// TIA Portal project "2020-10-30_TestMotoreNO_OK" (V16)

(* hardware
DEVICE "S7-1200 station_1"  S7-1200 Station
   slot 0: "Telaio di montaggio_0"  Rack  V1.0
   slot 1: "PLC_1"  CPU 1215C DC/DC/DC  6ES7 215-1AG40-0XB0  V4.2
*)

// ===== PLC "PLC_1"  CPU 1215C DC/DC/DC =====

VAR_GLOBAL   // PLC tag table "Tabella delle variabili standard"
   "finecorsa_NC" AT %I0.0 : Bool;
   "Presenza_tensione_NA" AT %I0.1 : Bool;
   "Ventilatore_motore_NA" AT %I0.3 : Bool;
   "Start_NA" AT %I0.5 : Bool;
   "Stop_NC" AT %I0.6 : Bool;
   "Allarme_NC" AT %I0.2 : Bool;
   "Ripristino_NA" AT %I0.7 : Bool;
   "Sensore termico mot_NA" AT %I0.4 : Bool;
   "Motore" AT %Q0.0 : Bool;
   "Allarme_mem" AT %Q0.1 : Bool;
   "M_IB0_NCNA" AT %MB0 : Byte;
   "Finecorsa" AT %M0.0 : Bool;
   "Presenza tensione" AT %M0.1 : Bool;
   "Ventilatore motore" AT %M0.3 : Bool;
   "Start" AT %M0.5 : Bool;
   "Stop" AT %M0.6 : Bool;
   "Allarme" AT %M0.2 : Bool;
   "Ripristino" AT %M0.7 : Bool;
   "Sempre_vera" AT %M6.0 : Bool;
   "Ingressi" AT %IB0 : Byte;
   "XXX_Start_old" AT %M1.5 : Bool;
   "XXX_Ripristino_old" AT %M1.7 : Bool;
   "Sensore_termico_mot" AT %M0.4 : Bool;
   "Guasto_ventil" AT %Q0.2 : Bool;
   "Allarme_gen" AT %Q0.3 : Bool;
   "Arresto_anomalo" AT %Q0.4 : Bool;
   "XXX2_ripristino_old" AT %M2.7 : Bool;
   "XXX2_start_old" AT %M2.5 : Bool;
END_VAR

VAR_GLOBAL CONSTANT   // PLC tag table "Tabella delle variabili standard"
   "Maschera NCNA" : Byte := 2#01000101;
END_VAR

ORGANIZATION_BLOCK "Main"   // OB1, LAD, ProgramCycle
TITLE = "Main Program Sweep (Cycle)"
{ S7_Optimized_Access := 'TRUE' }
VERSION : 0.1
// Programma c_mot_all_guast_arresto anomalo
// Step:
// a_ gestione start (I0.5 NA) Stop (I0.6 NC) motore (Q0.0) se presenza tensione (I0.1), con ventilatore acceso (I0.3 NA), logica di finecorsa di sicurezza (i0.0, NC) per arresto motore e sensore termico motore non intervenuto (I0.4 NA). Gestione Lampada Allarme (Q0.1) con memorizzazione ripristino e rientro (Allarme I0.2, NC, Ripristino I0.7 NA)
// 
// b_ funzionalità a, più gestione guasto ventilazione motore (Q0.2) se ventilatore acceso (I0.3 NA) e sensore termico motore intervenuto (I0.4 NA) con motore in movimento. 
// 
// c_ aggiunta gestione Allarme_generale (Q0.3), comprensivo di lampada allarme e guasto ventilatore, e aggiunta arresto motore anomalo (Q0.4) che si accende se il motore viene arrestato da situazioni non corrette (intervento finecorsa di sicurezza o allarme o caduta presenza tensione). Il pulsante Start viene utilizzato per resettare l'anomalia che è di sola segnalazione e non necessita di ripristino
// 
// ISTRUZIONI 
// *Si realizzi un programma di controllo per un motore. Il motore è azionato da un pulsante di Start e fermato dal pulsante di Stop.
// 
// Mappare ingressi NA/NC in memoria, in modo da lavorare in logica vera nel programma.
// Il motore parte se ho tensione, premo start e non sono in condizioni anomale per le quali il motore deve stare fermo.
// Il motore deve fermarsi se c'è un allarme o premo stop o finecorsa o se cade la tensione.
// Si consideri il fermo motore anche in caso di guasto ventilatore e e sensore termico
// 
// NOTA: Gestire incastro Pulsanti e motore
// 
// I0.0	Finecorsa_NC
// I0.1	Presenza_Tensione_NA
// I0.2	Allarme_NC	
// I0.3	Ventilatore_Motore_NA
// I0.4	Sensore_Termico_Motore_NA
// I0.5	Start_NA
// I0.6	Stop_NC
// I0.7	Ripristino_NA
// 
// Q0.0	Motore			   Motore avviato
// Q0.1	Lampada_Allarme	   Segnalazione allarme con memorizzazione ripristino e rientro
// Q0.2    Sirena guasto Ventilatore     Se Motore ON e Ventilatore ON e Sensore Termico ON allora Q0.3    Allarme_generale      Si setta in Presenza di Allarmemem o si guasto Ventil e si resetta con Ripristino
// Q0.4    Arresto motore anomalo     Si accende se il motore viene arrestato da situazioni non corrette (intervento finecorsa di sicurezza o allarme o caduta presenza tensione). Il pulsante Start viene utilizzato per resettare l'anomalia che è di sola segnalazione e non necessita di ripristino
   VAR_TEMP   // added for the SCL form of the ladder/FBD networks
      _w1 : Bool;
   END_VAR
BEGIN

REGION Network 1: Bit Sempre_vero
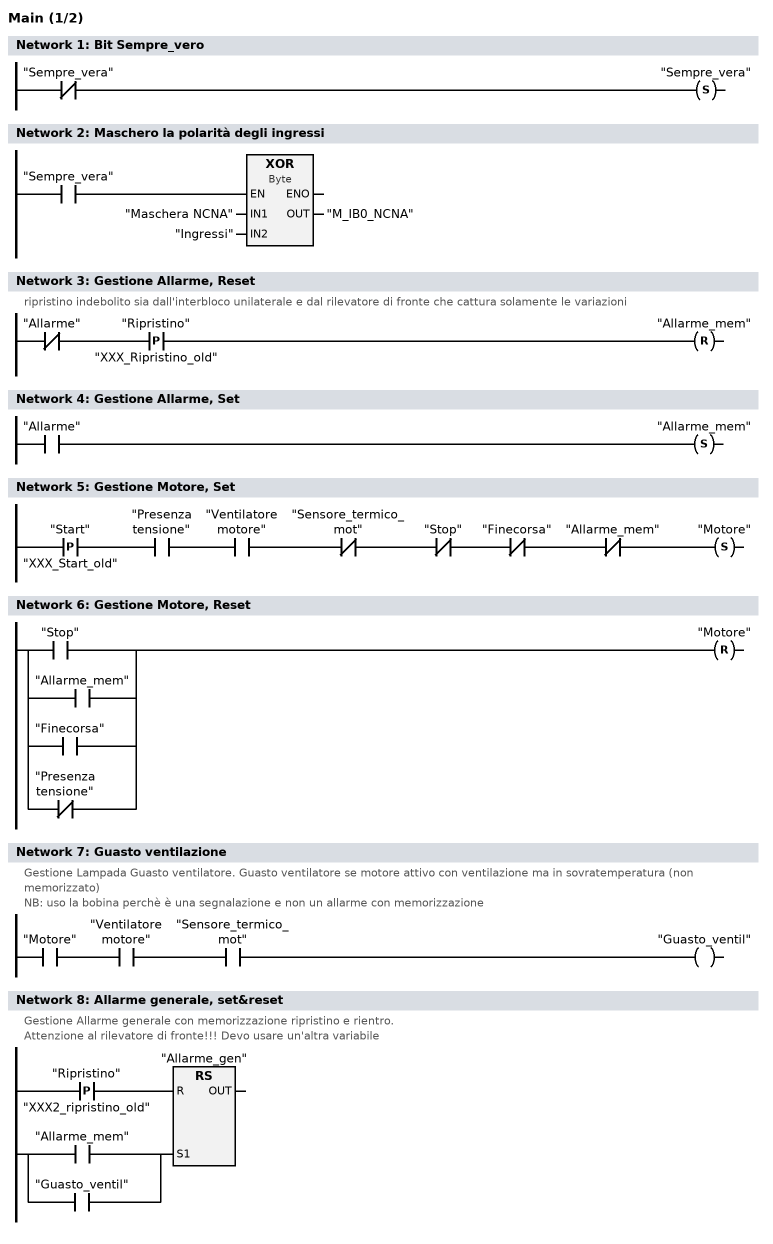
   RUNG wire#powerrail
      I_Contact( "Sempre_vera" )
      S_Coil( "Sempre_vera" )
   END_RUNG
   // the same network as SCL:
   IF NOT "Sempre_vera" THEN "Sempre_vera" := TRUE; END_IF;
END_REGION

REGION Network 2: Maschero la polarità degli ingressi
   IF "Sempre_vera" THEN "M_IB0_NCNA" := "Maschera NCNA" XOR "Ingressi"; END_IF;
END_REGION

REGION Network 3: Gestione Allarme, Reset
   // ripristino indebolito sia dall'interbloco unilaterale e dal rilevatore di fronte che cattura solamente le variazioni
   RUNG wire#powerrail
      I_Contact( "Allarme" )
      P_Contact(operand := "Ripristino", bit := "XXX_Ripristino_old")
      R_Coil( "Allarme_mem" )
   END_RUNG
   // the same network as SCL:
   #_w1 := NOT "Allarme" AND "Ripristino" AND NOT "XXX_Ripristino_old";   // rising edge of "Ripristino"
   "XXX_Ripristino_old" := "Ripristino";
   IF #_w1 THEN "Allarme_mem" := FALSE; END_IF;
END_REGION

REGION Network 4: Gestione Allarme, Set
   RUNG wire#powerrail
      Contact( "Allarme" )
      S_Coil( "Allarme_mem" )
   END_RUNG
   // the same network as SCL:
   IF "Allarme" THEN "Allarme_mem" := TRUE; END_IF;
END_REGION

REGION Network 5: Gestione Motore, Set
   RUNG wire#powerrail
      P_Contact(operand := "Start", bit := "XXX_Start_old")
      Contact( "Presenza tensione" )
      Contact( "Ventilatore motore" )
      I_Contact( "Sensore_termico_mot" )
      I_Contact( "Stop" )
      I_Contact( "Finecorsa" )
      I_Contact( "Allarme_mem" )
      S_Coil( "Motore" )
   END_RUNG
   // the same network as SCL:
   #_w1 := "Start" AND NOT "XXX_Start_old";   // rising edge of "Start"
   "XXX_Start_old" := "Start";
   IF #_w1 AND "Presenza tensione" AND "Ventilatore motore" AND NOT "Sensore_termico_mot" AND NOT "Stop" AND NOT "Finecorsa" AND NOT "Allarme_mem" THEN
       "Motore" := TRUE;
   END_IF;
END_REGION

REGION Network 6: Gestione Motore, Reset
   RUNG wire#powerrail
      Contact( "Stop" )
      wire#w1
      R_Coil( "Motore" )
   END_RUNG
   RUNG wire#powerrail
      Contact( "Allarme_mem" )
   END_RUNG wire#w1
   RUNG wire#powerrail
      Contact( "Finecorsa" )
   END_RUNG wire#w1
   RUNG wire#powerrail
      I_Contact( "Presenza tensione" )
   END_RUNG wire#w1
   // the same network as SCL:
   IF "Stop" OR "Allarme_mem" OR "Finecorsa" OR NOT "Presenza tensione" THEN "Motore" := FALSE; END_IF;
END_REGION

REGION Network 7: Guasto ventilazione
   // Gestione Lampada Guasto ventilatore. Guasto ventilatore se motore attivo con ventilazione ma in sovratemperatura (non memorizzato)
   // NB: uso la bobina perchè è una segnalazione e non un allarme con memorizzazione
   RUNG wire#powerrail
      Contact( "Motore" )
      Contact( "Ventilatore motore" )
      Contact( "Sensore_termico_mot" )
      Coil( "Guasto_ventil" )
   END_RUNG
   // the same network as SCL:
   "Guasto_ventil" := "Motore" AND "Ventilatore motore" AND "Sensore_termico_mot";
END_REGION

REGION Network 8: Allarme generale, set&reset
   // Gestione Allarme generale con memorizzazione ripristino e rientro.
   // Attenzione al rilevatore di fronte!!! Devo usare un'altra variabile
   RUNG wire#powerrail
      P_Contact(operand := "Ripristino", bit := "XXX2_ripristino_old")
      S_RS(operand := "Allarme_gen", s1 := wire#w1)
   END_RUNG
   RUNG wire#powerrail
      Contact( "Allarme_mem" )
   END_RUNG wire#w1
   RUNG wire#powerrail
      Contact( "Guasto_ventil" )
   END_RUNG wire#w1
   // the same network as SCL:
   #_w1 := "Ripristino" AND NOT "XXX2_ripristino_old";   // rising edge of "Ripristino"
   "XXX2_ripristino_old" := "Ripristino";
   IF #_w1 THEN
       "Allarme_gen" := FALSE;   // RS flip-flop
   END_IF;
   IF "Allarme_mem" OR "Guasto_ventil" THEN "Allarme_gen" := TRUE; END_IF;
END_REGION

REGION Network 9: Condizione arresto anomalo, reset
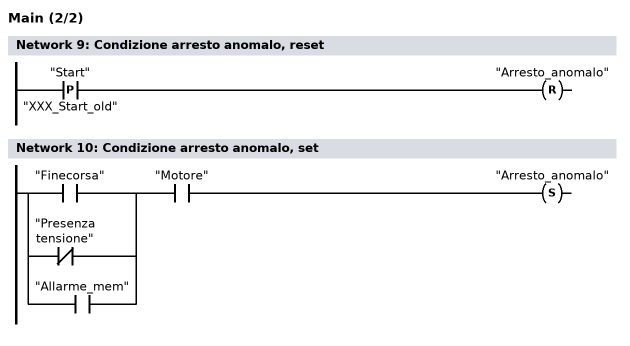
   RUNG wire#powerrail
      P_Contact(operand := "Start", bit := "XXX_Start_old")
      R_Coil( "Arresto_anomalo" )
   END_RUNG
   // the same network as SCL:
   #_w1 := "Start" AND NOT "XXX_Start_old";   // rising edge of "Start"
   "XXX_Start_old" := "Start";
   IF #_w1 THEN "Arresto_anomalo" := FALSE; END_IF;
END_REGION

REGION Network 10: Condizione arresto anomalo, set
   RUNG wire#powerrail
      Contact( "Finecorsa" )
      wire#w1
      Contact( "Motore" )
      S_Coil( "Arresto_anomalo" )
   END_RUNG
   RUNG wire#powerrail
      I_Contact( "Presenza tensione" )
   END_RUNG wire#w1
   RUNG wire#powerrail
      Contact( "Allarme_mem" )
   END_RUNG wire#w1
   // the same network as SCL:
   IF ("Finecorsa" OR NOT "Presenza tensione" OR "Allarme_mem") AND "Motore" THEN
       "Arresto_anomalo" := TRUE;
   END_IF;
END_REGION
END_ORGANIZATION_BLOCK